Omron CX-Programmer project NewProject (CX-Programmer 9.75)

# PLC NewPLC1: CPM1(CPM1A) CPU20

## Global symbols (name address type ; comment)
0.00 BOOL  ; Emergency
0.01 BOOL  ; Tempreture
0.02 BOOL  ; Emergency
0.03 BOOL  ; temp ok
0.04 BOOL  ; env1 arror
0.05 BOOL  ; env2 error
0.07 BOOL  ; Air Pressure
0.08 BOOL  ; Start Machine
0.09 BOOL  ; Stop Machine
0.10 BOOL  ; Man/Auto
10.00 BOOL  ; M1
10.00 BOOL  ; M1
10.01 BOOL  ; M2
10.02 BOOL  ; CLAMP
10.03 BOOL  ; Water Pump
10.04 BOOL  ; CLAMP
10.05 BOOL  ; Count Reached
10.06 BOOL  ; Allarm Lamp
10.07 BOOL  ; Machine OK
11.00 BOOL  ; Run Machine
11.01 BOOL  ; Automatic
11.02 BOOL  ; Manual
12.00 BOOL  ; Run M1 MANUALL
12.01 BOOL  ; Run M2 MANUALL
12.02 BOOL  ; Run Clamp MANUALL
12.03 BOOL  ; Run WATER PUMP MAN
13.00 BOOL  ; Run M1 AUTO
13.01 BOOL  ; Run M2 AUTO
13.02 BOOL  ; Run Clamp AUTO
15.00 BOOL  ; Cycle In progress
230 CHANNEL  ; HSC Channel 1
231 CHANNEL  ; HSC Channel 2
2.00 BOOL  ; Reset HSC
2.01 BOOL  ; Clamp Cycle
2.15 BOOL  ; reset hsc value on error
3.01 BOOL  ; clamp start
3.10 BOOL  ; Count Reached
4.00 BOOL  ; F1
4.01 BOOL  ; F2
4.02 BOOL  ; F3
4.03 BOOL  ; F4
4.04 BOOL  ; Reset Counter
4.04 BOOL  ; Reset Counter
5.00 BOOL  ; Reset Allarms
6.00 BOOL  ; F2 MAN
6.00 BOOL  ; F2 MAN
6.01 BOOL  ; F3 MAN
6.01 BOOL  ; F3 MAN
6.02 BOOL  ; F4 MAN
6.02 BOOL  ; F4 MAN
6.03 BOOL  ; F3&4 Man
7.00 BOOL  ; No Error
7.01 BOOL  ; Error
7.01 BOOL  ; Error
8.00 BOOL  ; Machine Ok
9.00 BOOL  ; InMain Menu Page
DM0 CHANNEL  ; Hmi page
DM100 CHANNEL  ; count set value
DM250 CHANNEL  ; HMI HSC SV
DM260 CHANNEL  ; HSC SV
DM50 CHANNEL  ; HSC PV1
DM501 CHANNEL  ; HMI HSC PV READ
DM50 CHANNEL  ; HSC PV1
DM51 CHANNEL  ; HSC PV2
DM60 CHANNEL  ; Count Present Value
HR0.00 BOOL  ; Emergency OK
HR0.01 BOOL  ; Tempreture Ok
HR0.01 BOOL  ; M2
HR0.02 BOOL  ; INV 1  M1 Error
HR0.02 BOOL  ; Clamp
HR0.03 BOOL  ; INV 2 M2 Error
HR0.04 BOOL  ; Air PS
HR2.00 BOOL  ; Encoder fault
HR2.01 BOOL  ; allarm Emergency
HR2.02 BOOL  ; allarm tempreture
HR2.03 BOOL  ; inv1 allarm
HR2.04 BOOL  ; inv2 allarm
HR2.05 BOOL  ; air pressure  allarm
HR5.00 BOOL  ; F1
HR5.01 BOOL  ; F2
HR5.02 BOOL  ; F3
HR5.03 BOOL  ; F4

## Program NewProgram1 (no task)

### Section Main
; Program designed by eng mahmoud shaban ahmed

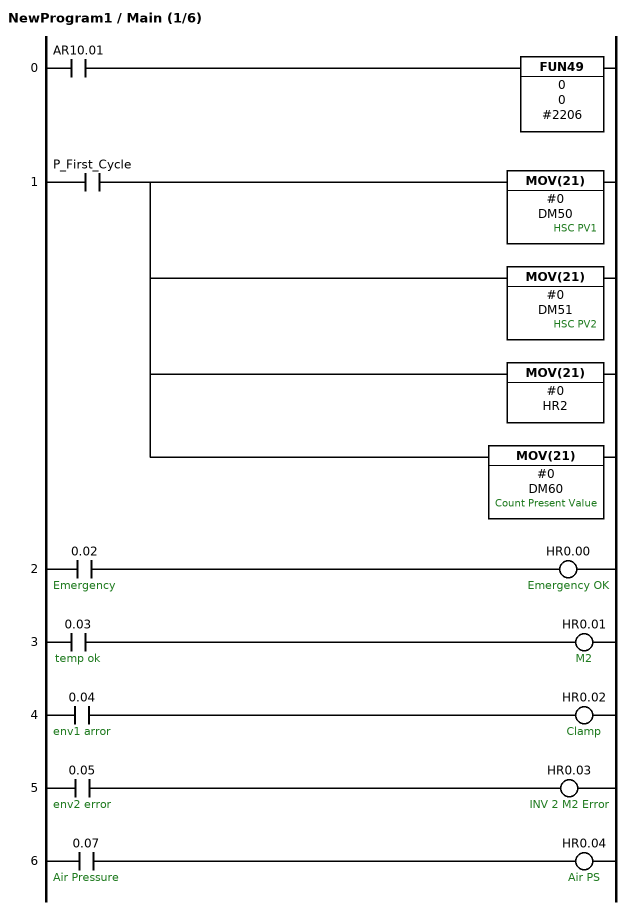
; rung 0
LD AR10.01
FUN49 0 0 #2206
; rung 1
LD P_First_Cycle
MOV(21) #0 DM50  ; HSC PV1
MOV(21) #0 DM51  ; HSC PV2
MOV(21) #0 HR2
MOV(21) #0 DM60  ; Count Present Value
; rung 2
LD 0.02  ; Emergency
OUT HR0.00  ; Emergency OK
; rung 3
LD 0.03  ; temp ok
OUT HR0.01  ; M2
; rung 4
LD 0.04  ; env1 arror
OUT HR0.02  ; Clamp
; rung 5
LD 0.05  ; env2 error
OUT HR0.03  ; INV 2 M2 Error
; rung 6
LD 0.07  ; Air Pressure
OUT HR0.04  ; Air PS

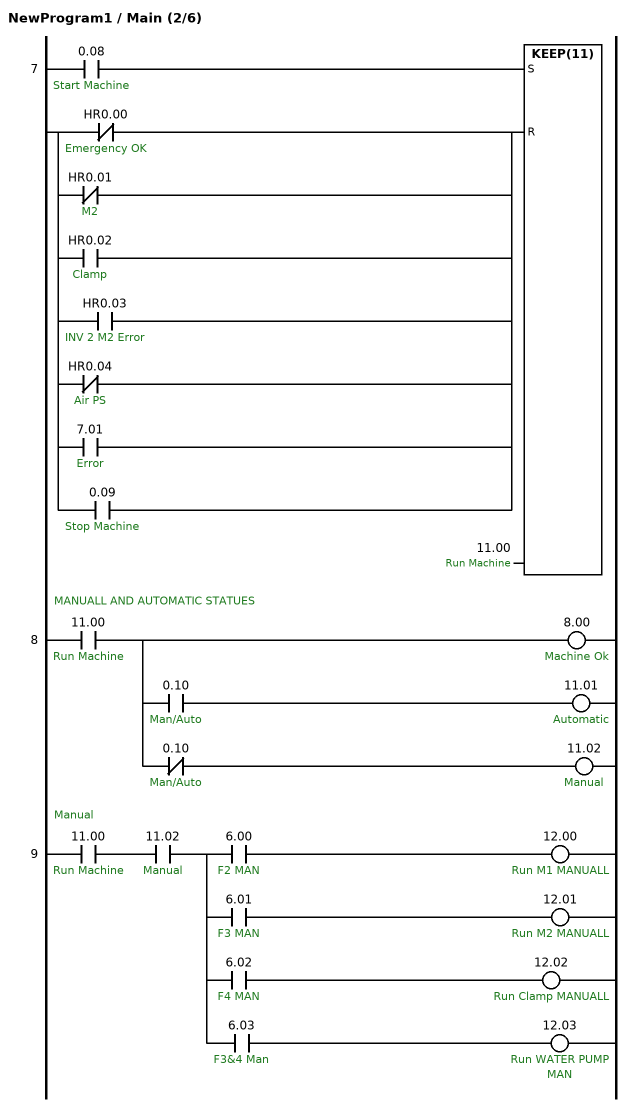
; rung 7
LD 0.08  ; Start Machine
LDNOT HR0.00  ; Emergency OK
ORNOT HR0.01  ; M2
OR HR0.02  ; Clamp
OR HR0.03  ; INV 2 M2 Error
ORNOT HR0.04  ; Air PS
OR 7.01  ; Error
OR 0.09  ; Stop Machine
KEEP(11) 11.00  ; Run Machine
; rung 8: MANUALL AND AUTOMATIC STATUES
LD 11.00  ; Run Machine
OUT TR0
OUT 8.00  ; Machine Ok
AND 0.10  ; Man/Auto
OUT 11.01  ; Automatic
LD TR0
ANDNOT 0.10  ; Man/Auto
OUT 11.02  ; Manual
; rung 9: Manual
LD 11.00  ; Run Machine
AND 11.02  ; Manual
OUT TR0
AND 6.00  ; F2 MAN
OUT 12.00  ; Run M1 MANUALL
LD TR0
AND 6.01  ; F3 MAN
OUT 12.01  ; Run M2 MANUALL
LD TR0
AND 6.02  ; F4 MAN
OUT 12.02  ; Run Clamp MANUALL
LD TR0
AND 6.03  ; F3&4 Man
OUT 12.03  ; Run WATER PUMP MAN

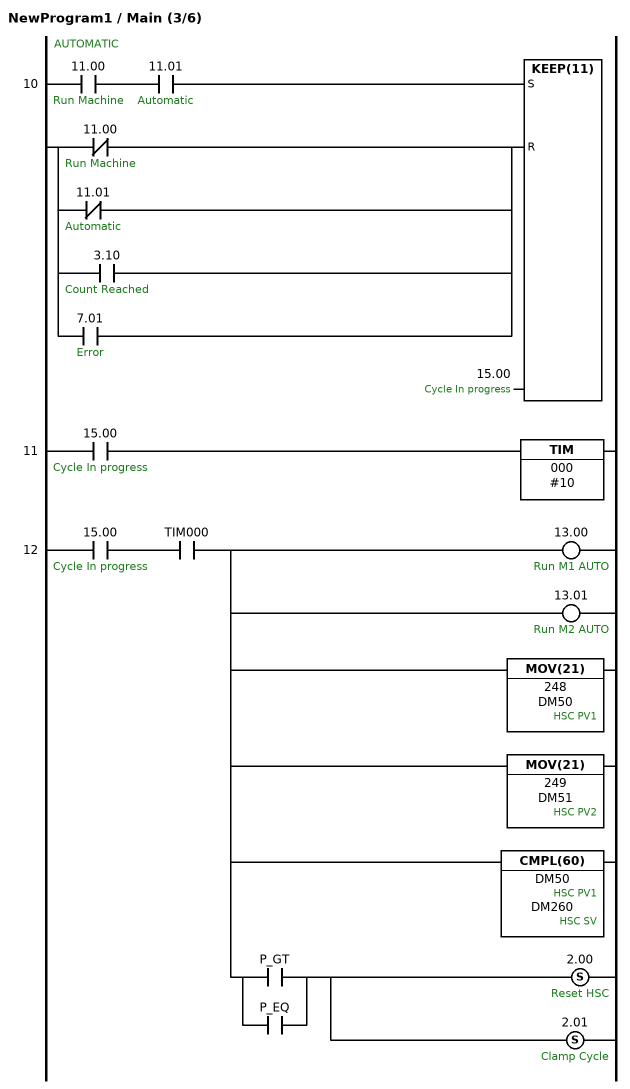
; rung 10: AUTOMATIC
LD 11.00  ; Run Machine
AND 11.01  ; Automatic
LDNOT 11.00  ; Run Machine
ORNOT 11.01  ; Automatic
OR 3.10  ; Count Reached
OR 7.01  ; Error
KEEP(11) 15.00  ; Cycle In progress
; rung 11
LD 15.00  ; Cycle In progress
TIM 000 #10
; rung 12
LD 15.00  ; Cycle In progress
AND TIM000
OUT 13.00  ; Run M1 AUTO
OUT 13.01  ; Run M2 AUTO
MOV(21) 248 DM50  ; HSC PV1
MOV(21) 249 DM51  ; HSC PV2
CMPL(60) DM50 DM260  ; HSC PV1, HSC SV
LD P_GT
OR P_EQ
ANDLD
SET 2.00  ; Reset HSC
SET 2.01  ; Clamp Cycle

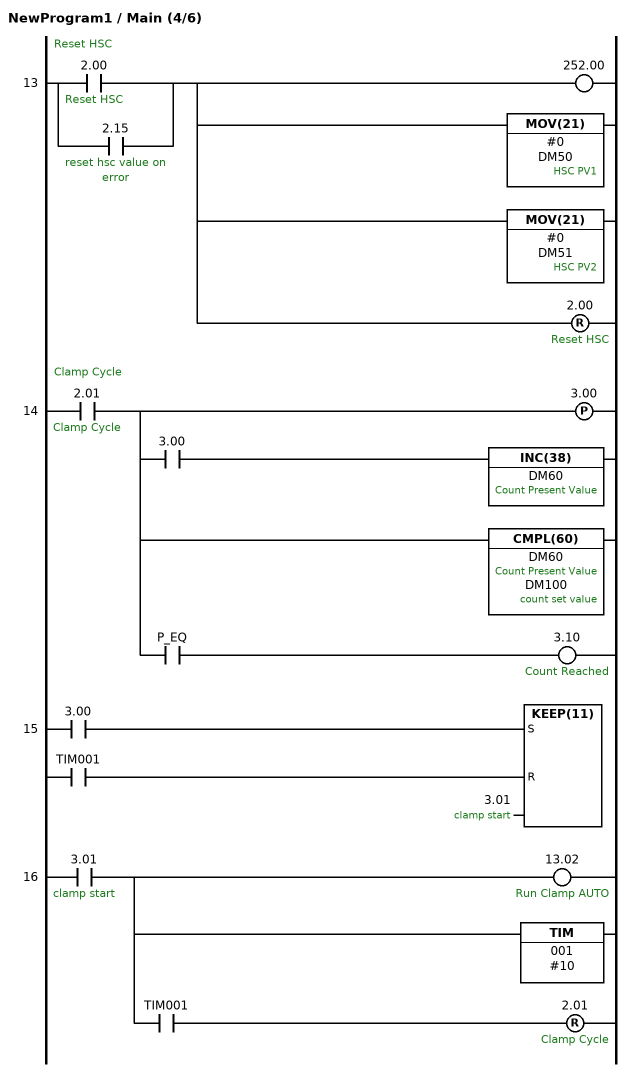
; rung 13: Reset HSC
LD 2.00  ; Reset HSC
OR 2.15  ; reset hsc value on error
OUT 252.00
MOV(21) #0 DM50  ; HSC PV1
MOV(21) #0 DM51  ; HSC PV2
RSET 2.00  ; Reset HSC
; rung 14: Clamp Cycle
LD 2.01  ; Clamp Cycle
OUT TR0
DIFU(13) 3.00
AND 3.00
INC(38) DM60  ; Count Present Value
LD TR0
CMPL(60) DM60 DM100  ; Count Present Value, count set value
AND P_EQ
OUT 3.10  ; Count Reached
; rung 15
LD 3.00
LD TIM001
KEEP(11) 3.01  ; clamp start
; rung 16
LD 3.01  ; clamp start
OUT 13.02  ; Run Clamp AUTO
TIM 001 #10
AND TIM001
RSET 2.01  ; Clamp Cycle

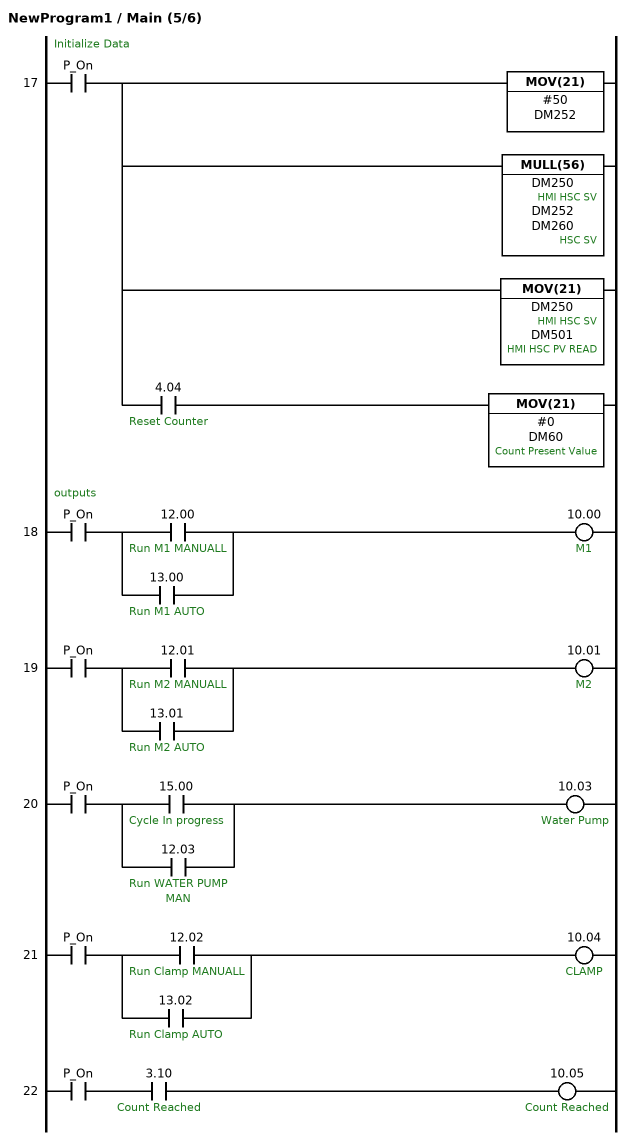
; rung 17: Initialize Data
LD P_On
MOV(21) #50 DM252
MULL(56) DM250 DM252 DM260  ; HMI HSC SV, HSC SV
MOV(21) DM250 DM501  ; HMI HSC SV, HMI HSC PV READ
AND 4.04  ; Reset Counter
MOV(21) #0 DM60  ; Count Present Value
; rung 18: outputs
LD P_On
LD 12.00  ; Run M1 MANUALL
OR 13.00  ; Run M1 AUTO
ANDLD
OUT 10.00  ; M1
; rung 19
LD P_On
LD 12.01  ; Run M2 MANUALL
OR 13.01  ; Run M2 AUTO
ANDLD
OUT 10.01  ; M2
; rung 20
LD P_On
LD 15.00  ; Cycle In progress
OR 12.03  ; Run WATER PUMP MAN
ANDLD
OUT 10.03  ; Water Pump
; rung 21
LD P_On
LD 12.02  ; Run Clamp MANUALL
OR 13.02  ; Run Clamp AUTO
ANDLD
OUT 10.04  ; CLAMP
; rung 22
LD P_On
AND 3.10  ; Count Reached
OUT 10.05  ; Count Reached

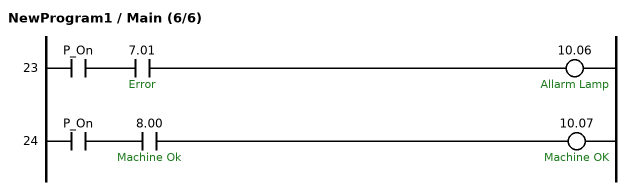
; rung 23
LD P_On
AND 7.01  ; Error
OUT 10.06  ; Allarm Lamp
; rung 24
LD P_On
AND 8.00  ; Machine Ok
OUT 10.07  ; Machine OK

### Section HMI

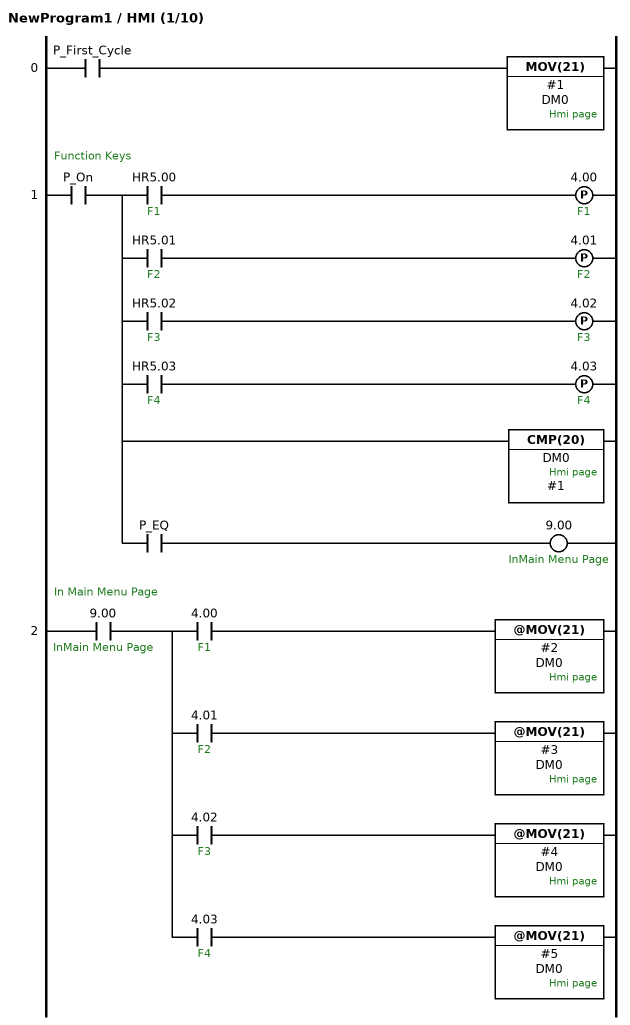
; rung 0
LD P_First_Cycle
MOV(21) #1 DM0  ; Hmi page
; rung 1: Function Keys
LD P_On
OUT TR0
AND HR5.00  ; F1
DIFU(13) 4.00  ; F1
LD TR0
AND HR5.01  ; F2
DIFU(13) 4.01  ; F2
LD TR0
AND HR5.02  ; F3
DIFU(13) 4.02  ; F3
LD TR0
AND HR5.03  ; F4
DIFU(13) 4.03  ; F4
LD TR0
CMP(20) DM0 #1  ; Hmi page
AND P_EQ
OUT 9.00  ; InMain Menu Page
; rung 2: In Main Menu Page
LD 9.00  ; InMain Menu Page
OUT TR0
AND 4.00  ; F1
@MOV(21) #2 DM0  ; Hmi page  // Main Page
LD TR0
AND 4.01  ; F2
@MOV(21) #3 DM0  ; Hmi page  // parameter page
LD TR0
AND 4.02  ; F3
@MOV(21) #4 DM0  ; Hmi page  // Allarm Page
LD TR0
AND 4.03  ; F4
@MOV(21) #5 DM0  ; Hmi page  // Manuall page

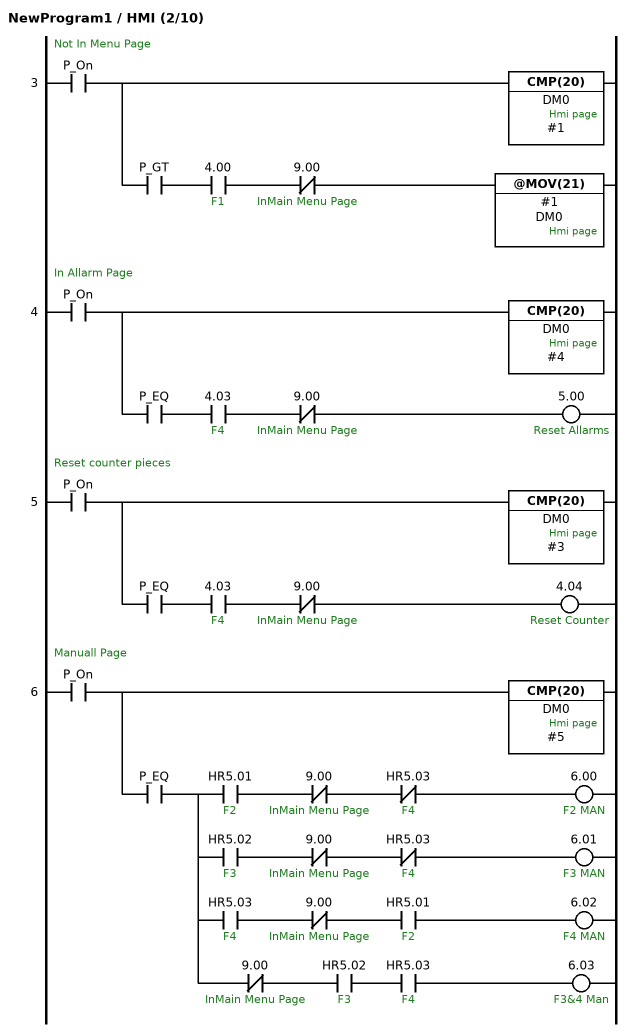
; rung 3: Not In Menu Page
LD P_On
CMP(20) DM0 #1  ; Hmi page  // If the page number greter than 1 and press F1 return to page 1
AND P_GT
AND 4.00  ; F1
ANDNOT 9.00  ; InMain Menu Page
@MOV(21) #1 DM0  ; Hmi page
; rung 4: In Allarm Page
LD P_On
CMP(20) DM0 #4  ; Hmi page  // If the page number 4 and press F4 reset all allarms
AND P_EQ
AND 4.03  ; F4
ANDNOT 9.00  ; InMain Menu Page
OUT 5.00  ; Reset Allarms
; rung 5: Reset counter pieces
LD P_On
CMP(20) DM0 #3  ; Hmi page  // If the page number  3 and press F4 Reset counter
AND P_EQ
AND 4.03  ; F4
ANDNOT 9.00  ; InMain Menu Page
OUT 4.04  ; Reset Counter
; rung 6: Manuall Page
LD P_On
CMP(20) DM0 #5  ; Hmi page  // If the page number  3 and press F4 Reset counter
AND P_EQ
OUT TR0
AND HR5.01  ; F2
ANDNOT 9.00  ; InMain Menu Page
ANDNOT HR5.03  ; F4
OUT 6.00  ; F2 MAN
LD TR0
AND HR5.02  ; F3
ANDNOT 9.00  ; InMain Menu Page
ANDNOT HR5.03  ; F4
OUT 6.01  ; F3 MAN
LD TR0
AND HR5.03  ; F4
ANDNOT 9.00  ; InMain Menu Page
AND HR5.01  ; F2
OUT 6.02  ; F4 MAN
LD TR0
ANDNOT 9.00  ; InMain Menu Page
AND HR5.02  ; F3
AND HR5.03  ; F4
OUT 6.03  ; F3&4 Man

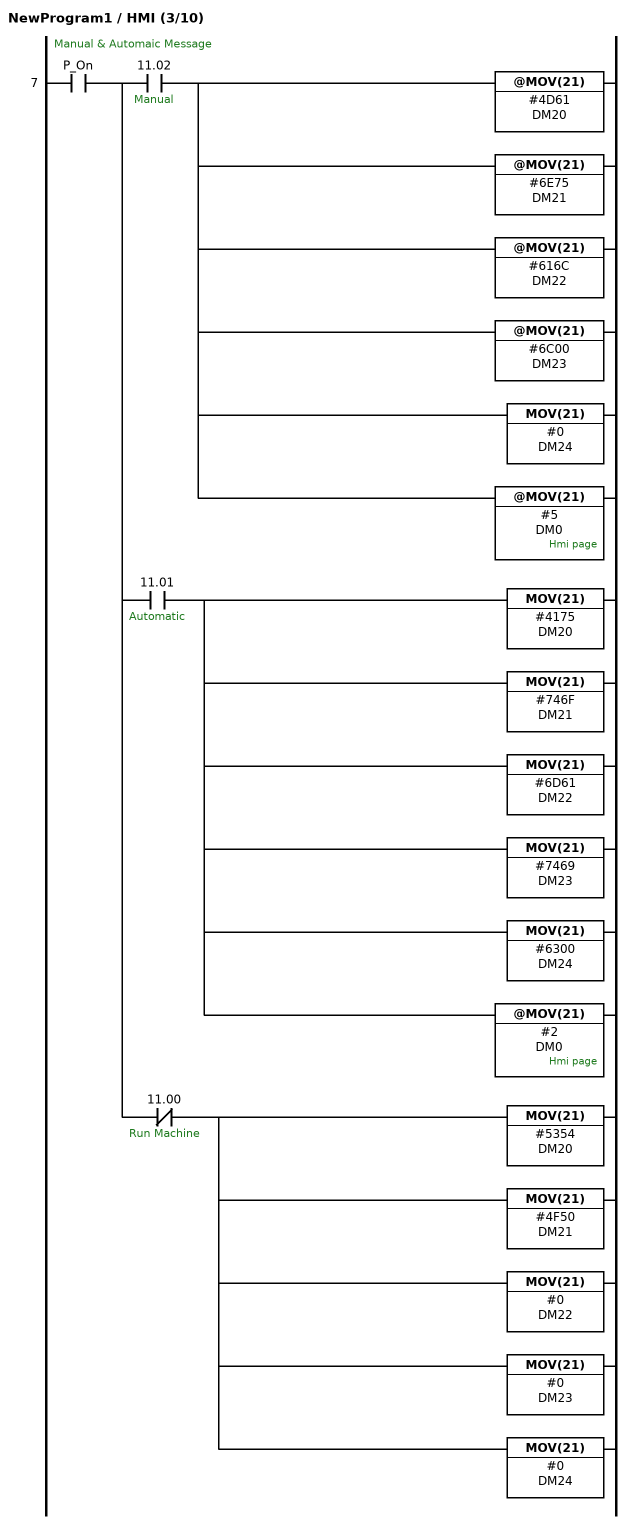
; rung 7: Manual & Automaic Message
LD P_On
OUT TR0
AND 11.02  ; Manual
@MOV(21) #4D61 DM20
@MOV(21) #6E75 DM21
@MOV(21) #616C DM22
@MOV(21) #6C00 DM23
MOV(21) #0 DM24
@MOV(21) #5 DM0  ; Hmi page
LD TR0
AND 11.01  ; Automatic
MOV(21) #4175 DM20
MOV(21) #746F DM21
MOV(21) #6D61 DM22
MOV(21) #7469 DM23
MOV(21) #6300 DM24
@MOV(21) #2 DM0  ; Hmi page
LD TR0
ANDNOT 11.00  ; Run Machine
MOV(21) #5354 DM20  // MACHINE STOP MESSAGE
MOV(21) #4F50 DM21
MOV(21) #0 DM22
MOV(21) #0 DM23
MOV(21) #0 DM24

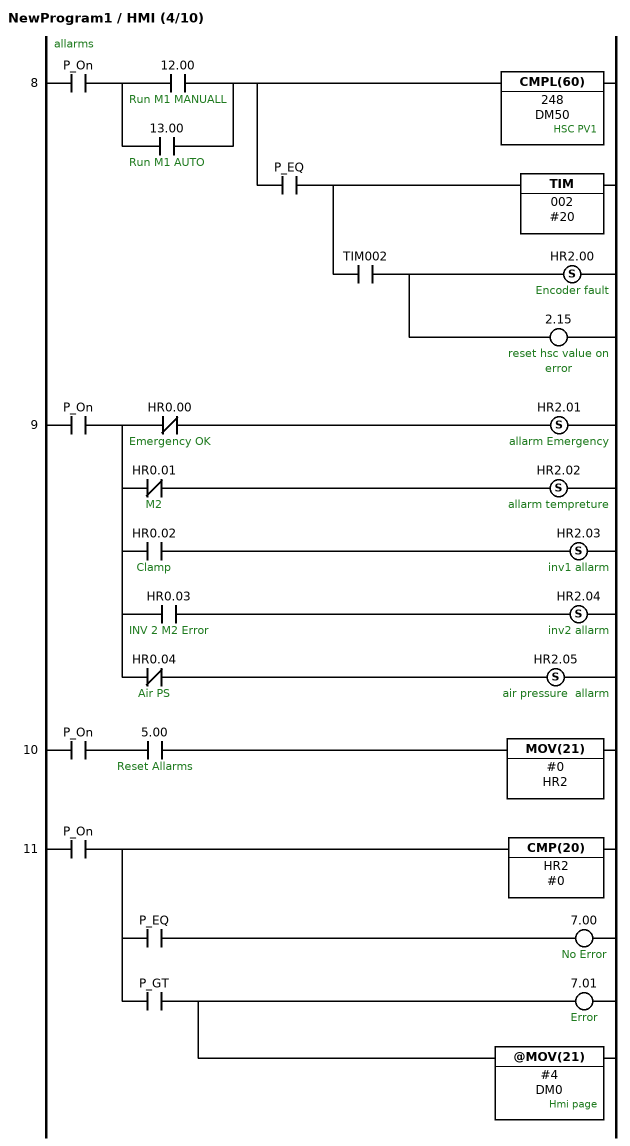
; rung 8: allarms
LD P_On
LD 12.00  ; Run M1 MANUALL
OR 13.00  ; Run M1 AUTO
ANDLD
CMPL(60) 248 DM50  ; HSC PV1
AND P_EQ
TIM 002 #20
AND TIM002
SET HR2.00  ; Encoder fault
OUT 2.15  ; reset hsc value on error
; rung 9
LD P_On
OUT TR0
ANDNOT HR0.00  ; Emergency OK
SET HR2.01  ; allarm Emergency
LD TR0
ANDNOT HR0.01  ; M2
SET HR2.02  ; allarm tempreture
LD TR0
AND HR0.02  ; Clamp
SET HR2.03  ; inv1 allarm
LD TR0
AND HR0.03  ; INV 2 M2 Error
SET HR2.04  ; inv2 allarm
LD TR0
ANDNOT HR0.04  ; Air PS
SET HR2.05  ; air pressure  allarm
; rung 10
LD P_On
AND 5.00  ; Reset Allarms
MOV(21) #0 HR2
; rung 11
LD P_On
OUT TR0
CMP(20) HR2 #0
AND P_EQ
OUT 7.00  ; No Error
LD TR0
AND P_GT
OUT 7.01  ; Error
@MOV(21) #4 DM0  ; Hmi page

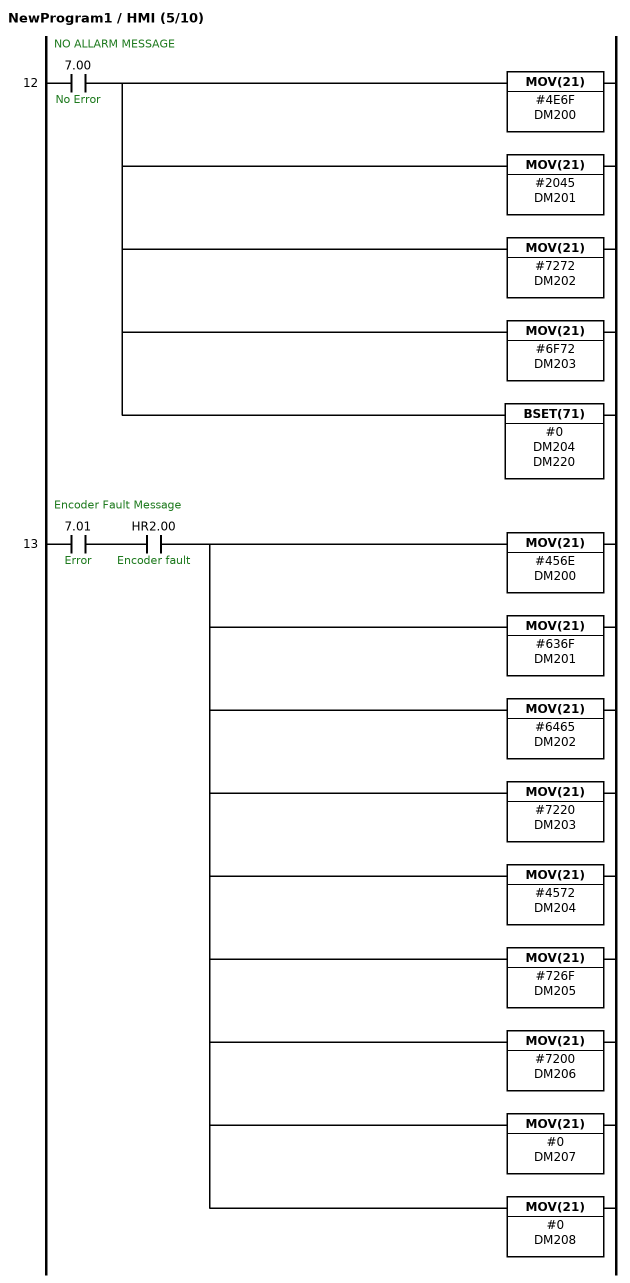
; rung 12: NO ALLARM MESSAGE
LD 7.00  ; No Error
MOV(21) #4E6F DM200
MOV(21) #2045 DM201
MOV(21) #7272 DM202
MOV(21) #6F72 DM203
BSET(71) #0 DM204 DM220
; rung 13: Encoder Fault Message
LD 7.01  ; Error
AND HR2.00  ; Encoder fault
MOV(21) #456E DM200
MOV(21) #636F DM201
MOV(21) #6465 DM202
MOV(21) #7220 DM203
MOV(21) #4572 DM204
MOV(21) #726F DM205
MOV(21) #7200 DM206
MOV(21) #0 DM207
MOV(21) #0 DM208

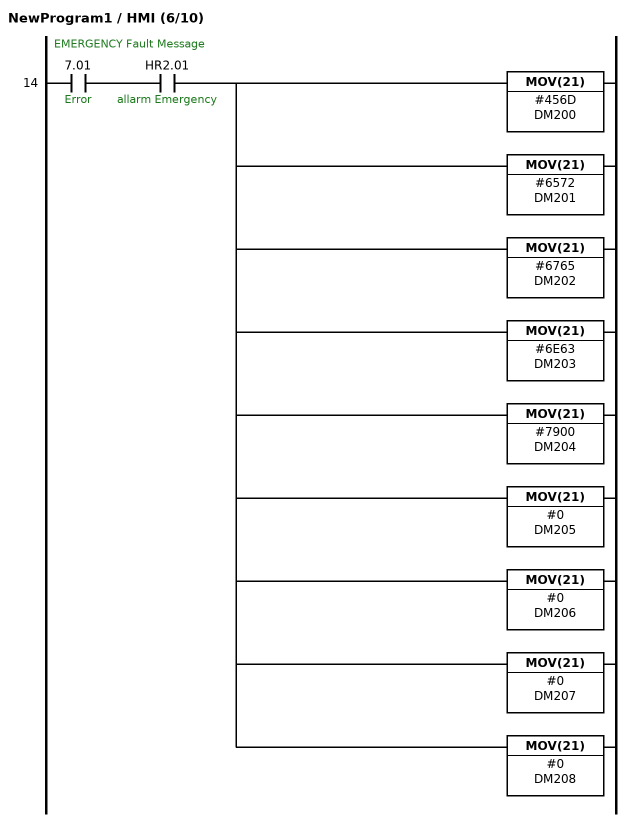
; rung 14: EMERGENCY Fault Message
LD 7.01  ; Error
AND HR2.01  ; allarm Emergency
MOV(21) #456D DM200
MOV(21) #6572 DM201
MOV(21) #6765 DM202
MOV(21) #6E63 DM203
MOV(21) #7900 DM204
MOV(21) #0 DM205
MOV(21) #0 DM206
MOV(21) #0 DM207
MOV(21) #0 DM208

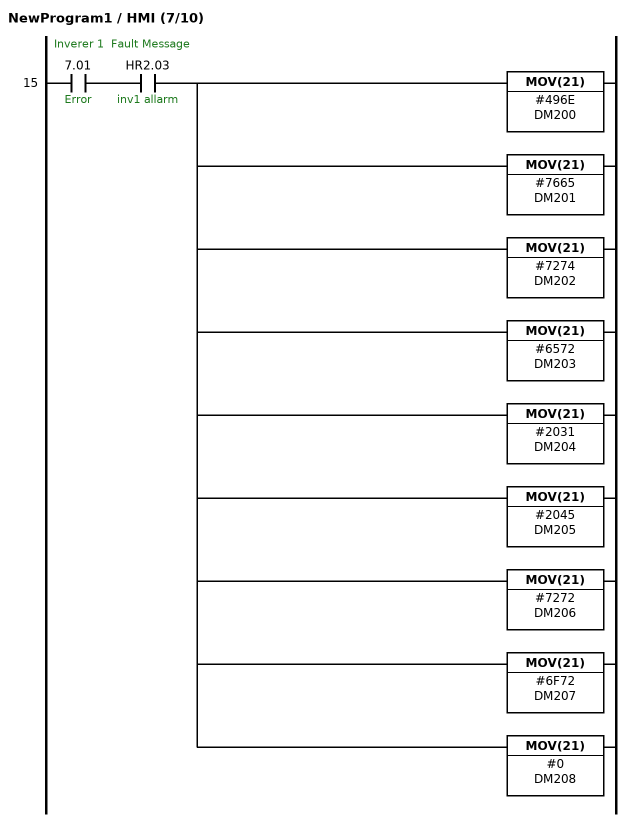
; rung 15: Inverer 1  Fault Message
LD 7.01  ; Error
AND HR2.03  ; inv1 allarm
MOV(21) #496E DM200
MOV(21) #7665 DM201
MOV(21) #7274 DM202
MOV(21) #6572 DM203
MOV(21) #2031 DM204
MOV(21) #2045 DM205
MOV(21) #7272 DM206
MOV(21) #6F72 DM207
MOV(21) #0 DM208

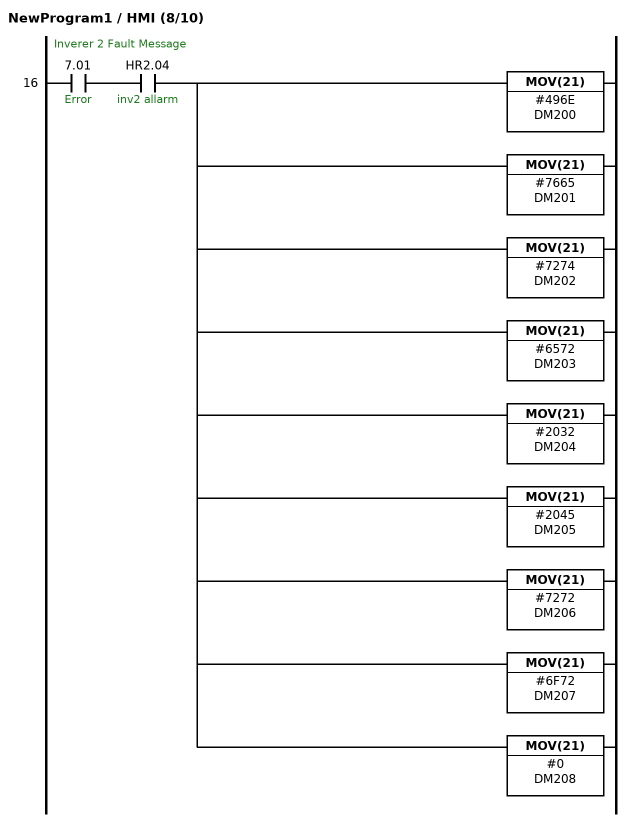
; rung 16: Inverer 2 Fault Message
LD 7.01  ; Error
AND HR2.04  ; inv2 allarm
MOV(21) #496E DM200
MOV(21) #7665 DM201
MOV(21) #7274 DM202
MOV(21) #6572 DM203
MOV(21) #2032 DM204
MOV(21) #2045 DM205
MOV(21) #7272 DM206
MOV(21) #6F72 DM207
MOV(21) #0 DM208

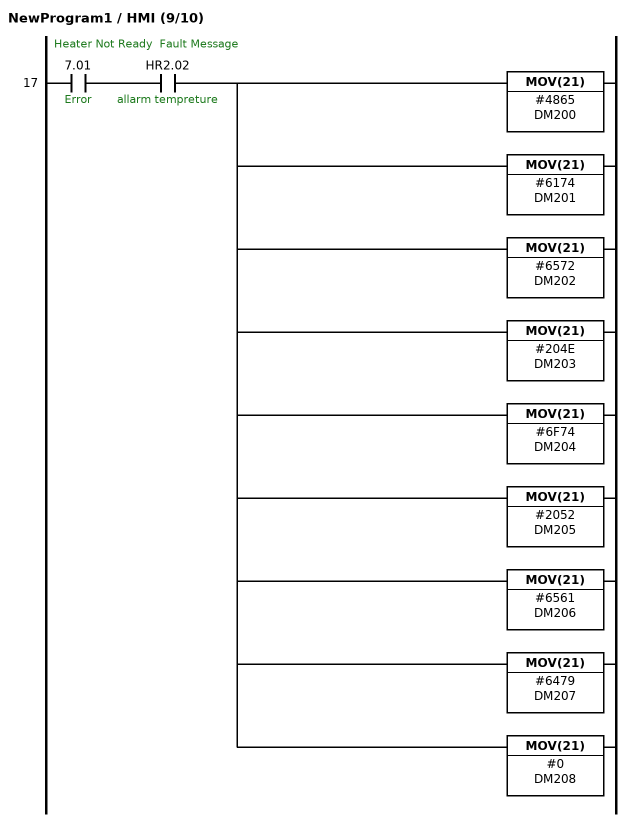
; rung 17: Heater Not Ready  Fault Message
LD 7.01  ; Error
AND HR2.02  ; allarm tempreture
MOV(21) #4865 DM200
MOV(21) #6174 DM201
MOV(21) #6572 DM202
MOV(21) #204E DM203
MOV(21) #6F74 DM204
MOV(21) #2052 DM205
MOV(21) #6561 DM206
MOV(21) #6479 DM207
MOV(21) #0 DM208

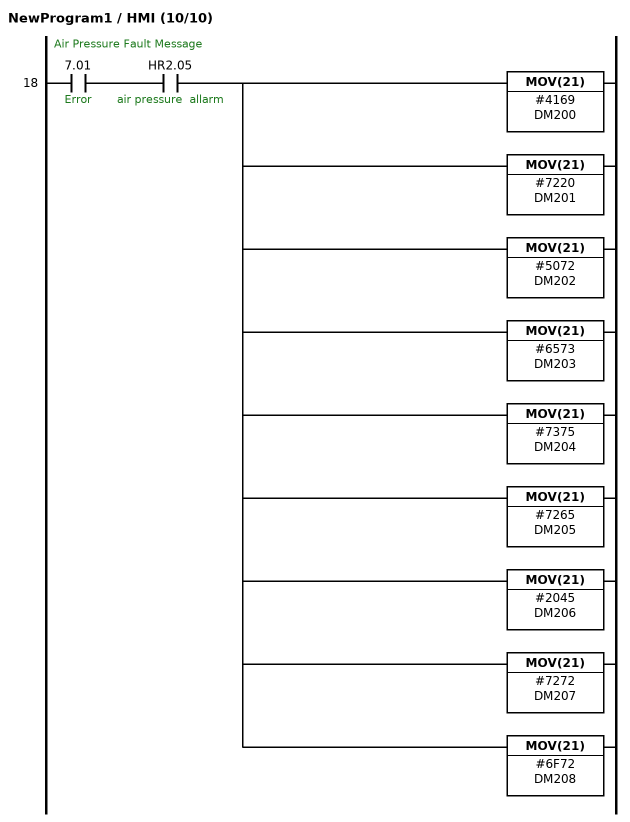
; rung 18: Air Pressure Fault Message
LD 7.01  ; Error
AND HR2.05  ; air pressure  allarm
MOV(21) #4169 DM200
MOV(21) #7220 DM201
MOV(21) #5072 DM202
MOV(21) #6573 DM203
MOV(21) #7375 DM204
MOV(21) #7265 DM205
MOV(21) #2045 DM206
MOV(21) #7272 DM207
MOV(21) #6F72 DM208

### Section END
; rung 0
END(01)